// TIA Portal V21 export
DATA_BLOCK "BatchRe"   // DB33
{ S7_Optimized_Access := 'TRUE' }
// stored: AutoNumber false, MemoryReserve 100
   VAR
      ReBit : Array[0..20] of Bool;
      BatchLinePrint : Array[0..60] of String;
   END_VAR
BEGIN
   BatchLinePrint[1] := 'BATCH STARTED';
   BatchLinePrint[2] := 'BATCH OVER';
   BatchLinePrint[3] := 'FILL WFI STARTED';
   BatchLinePrint[4] := 'FILL WFI PAUSED';
   BatchLinePrint[5] := 'FILL WFI RESUMED';
   BatchLinePrint[6] := 'FILL WFI OVER';
   BatchLinePrint[7] := 'FILL WFI RESET';
   BatchLinePrint[8] := 'TEMPERATURE CONTROL HEATING STARTED';
   BatchLinePrint[9] := 'TEMPERATURE CONTROL COOLING STARTED';
   BatchLinePrint[10] := 'TEMPERATURE CONTROL PAUSED';
   BatchLinePrint[11] := 'TEMPERATURE CONTROL RESUMED';
   BatchLinePrint[12] := 'TEMPERATURE CONTROL HEATING REACHED';
   BatchLinePrint[13] := 'TEMPERATURE CONTROL RESET';
   BatchLinePrint[14] := 'MM01 MIXING STARTED';
   BatchLinePrint[15] := 'MM01 MIXING PAUSED';
   BatchLinePrint[16] := 'MM01 MIXING RESUMED';
   BatchLinePrint[17] := 'MM01 MIXING OVER';
   BatchLinePrint[18] := 'MM01 MIXING RESET';
   BatchLinePrint[19] := 'PRODUCT RECIRCULATION STARTED';
   BatchLinePrint[20] := 'PRODUCT RECIRCULATION PAUSED';
   BatchLinePrint[21] := 'PRODUCT RECIRCULATION RESUMED';
   BatchLinePrint[22] := 'PRODUCT RECIRCULATION OVER';
   BatchLinePrint[23] := 'PRODUCT RECIRCULATION RESET';
   BatchLinePrint[24] := 'MANUAL RM ADDITION STARTED';
   BatchLinePrint[25] := 'MANUAL RM ADDITION PAUSED';
   BatchLinePrint[26] := 'MANUAL RM ADDITION RESUMED';
   BatchLinePrint[27] := 'MANUAL RM ADDITION OVER';
   BatchLinePrint[28] := 'MANUAL RM ADDITION RESET';
   BatchLinePrint[29] := 'N2 SPARGING STARTED';
   BatchLinePrint[30] := 'N2 SPARGING PAUSED';
   BatchLinePrint[31] := 'N2 SPARGING RESUMED';
   BatchLinePrint[32] := 'N2 SPARGING OVER';
   BatchLinePrint[33] := 'N2 SPARGING RESET';
   BatchLinePrint[34] := 'GAS BLANKETING STARTED';
   BatchLinePrint[35] := 'GAS BLANKETING PAUSED';
   BatchLinePrint[36] := 'GAS BLANKETING RESUMED';
   BatchLinePrint[37] := 'GAS BLANKETING RESET';
   BatchLinePrint[38] := 'FINAL VOLUME MAKEUP STARTED';
   BatchLinePrint[39] := 'FINAL VOLUME MAKEUP PAUSED';
   BatchLinePrint[40] := 'FINAL VOLUME MAKEUP RESUMED';
   BatchLinePrint[41] := 'FINAL VOLUME MAKEUP OVER';
   BatchLinePrint[42] := 'FINAL VOLUME MAKEUP RESET';
   BatchLinePrint[43] := 'PRODUCT TRANSFER STARTED';
   BatchLinePrint[44] := 'PRODUCT TRANSFER PAUSED';
   BatchLinePrint[45] := 'PRODUCT TRANSFER RESUMED';
   BatchLinePrint[46] := 'PRODUCT TRANSFER OVER';
   BatchLinePrint[47] := 'PRODUCT TRANSFER RESET';
   BatchLinePrint[48] := 'JACKET VENT OPEN';
   BatchLinePrint[49] := 'JACKET VENT CLOSE';
   BatchLinePrint[50] := 'JACKET DRAIN OPEN';
   BatchLinePrint[51] := 'JACKET DRAIN CLOSE';
   BatchLinePrint[52] := 'TEMPERATURE CONTROL COOLING REACHED';
   BatchLinePrint[53] := '-';
END_DATA_BLOCK
